PROGRAM MAIN
VAR
END_VAR

END_PROGRAM

(* stored: Version 1.1.0.1
   POU MAIN: Id {7ef286e7-0e39-40a6-9bda-8d5410adf0eb} *)
